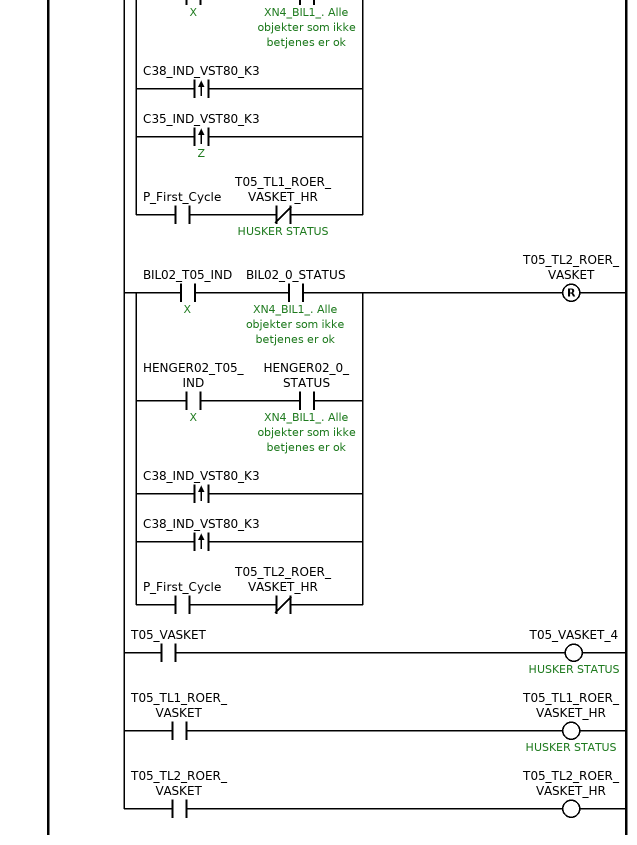
; [picture p936: NewProgram1 / T05_STATUS, rungs 1-1]
; rung 1: TANKOMRÅDET VASKET
LD P_On
OUT TR0
AND K3_TR23_TID_S
OUT TR1
LD C14_IND_VST80_K3  ; Z
OR C38_IND_VST80_K3
LD P_First_Cycle
AND T05_VASKET_4  ; HUSKER STATUS
ORLD
ANDLD
SET T05_VASKET
LD TR1
LD C38_IND_VST80_K3
OR C35_IND_VST80_K3  ; Z
LD P_First_Cycle
AND T05_TL1_ROER_VASKET_HR  ; HUSKER STATUS
ORLD
ANDLD
SET T05_TL1_ROER_VASKET
LD TR1
LD C38_IND_VST80_K3
OR C35_IND_VST80_K3  ; Z
LD P_First_Cycle
AND T05_TL2_ROER_VASKET_HR
ORLD
ANDLD
SET T05_TL2_ROER_VASKET
LD TR0
LD BIL01_T05_IND  ; X
AND BIL01_0_STATUS  ; XN4_BIL1_. Alle objekter som ikke betjenes er ok
LD HENGER01_T05_IND  ; X
AND HENGER01_0_STATUS  ; XN4_BIL1_. Alle objekter som ikke betjenes er ok
ORLD
LD BIL02_T05_IND  ; X
AND BIL02_0_STATUS  ; XN4_BIL1_. Alle objekter som ikke betjenes er ok
ORLD
LD HENGER02_T05_IND  ; X
AND HENGER02_0_STATUS  ; XN4_BIL1_. Alle objekter som ikke betjenes er ok
ORLD
@OR C38_IND_VST80_K3
@OR C14_IND_VST80_K3  ; Z
LD P_First_Cycle
ANDNOT T05_VASKET_4  ; HUSKER STATUS
ORLD
ANDLD
RSET T05_VASKET
LD TR0
LD BIL01_T05_IND  ; X
AND BIL01_0_STATUS  ; XN4_BIL1_. Alle objekter som ikke betjenes er ok
LD HENGER01_T05_IND  ; X
AND HENGER01_0_STATUS  ; XN4_BIL1_. Alle objekter som ikke betjenes er ok
ORLD
@OR C38_IND_VST80_K3
@OR C35_IND_VST80_K3  ; Z
LD P_First_Cycle
ANDNOT T05_TL1_ROER_VASKET_HR  ; HUSKER STATUS
ORLD
ANDLD
RSET T05_TL1_ROER_VASKET
LD TR0
LD BIL02_T05_IND  ; X
AND BIL02_0_STATUS  ; XN4_BIL1_. Alle objekter som ikke betjenes er ok
LD HENGER02_T05_IND  ; X
AND HENGER02_0_STATUS  ; XN4_BIL1_. Alle objekter som ikke betjenes er ok
ORLD
@OR C38_IND_VST80_K3
@OR C38_IND_VST80_K3
LD P_First_Cycle
ANDNOT T05_TL2_ROER_VASKET_HR
ORLD
ANDLD
RSET T05_TL2_ROER_VASKET
LD TR0
AND T05_VASKET
OUT T05_VASKET_4  ; HUSKER STATUS
LD TR0
AND T05_TL1_ROER_VASKET
OUT T05_TL1_ROER_VASKET_HR  ; HUSKER STATUS
LD TR0
AND T05_TL2_ROER_VASKET
OUT T05_TL2_ROER_VASKET_HR

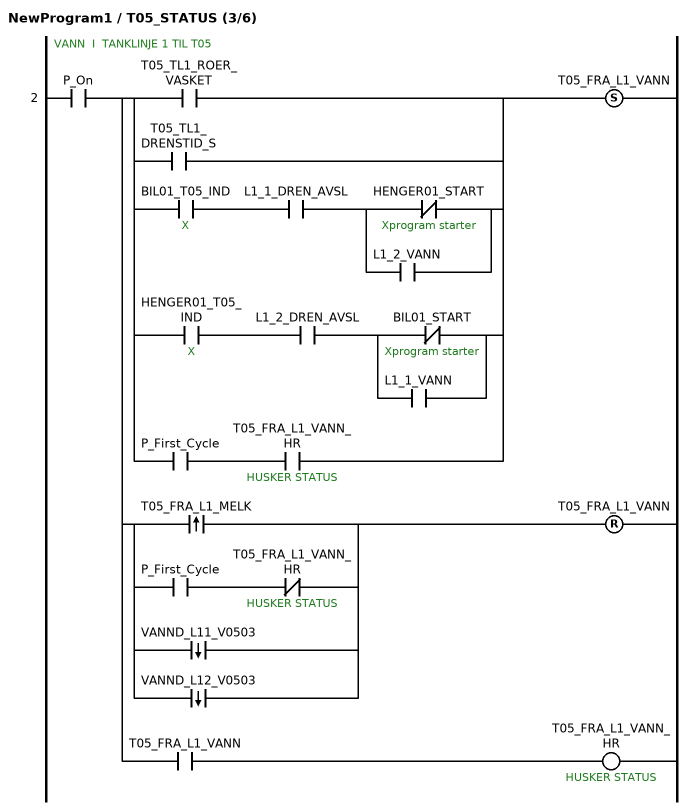
; rung 2: VANN  I  TANKLINJE 1 TIL T05
LD P_On
OUT TR0
LD T05_TL1_ROER_VASKET
OR T05_TL1_DRENSTID_S
LD BIL01_T05_IND  ; X
AND L1_1_DREN_AVSL
LDNOT HENGER01_START  ; Xprogram starter
OR L1_2_VANN
ANDLD
ORLD
LD HENGER01_T05_IND  ; X
AND L1_2_DREN_AVSL
LDNOT BIL01_START  ; Xprogram starter
OR L1_1_VANN
ANDLD
ORLD
LD P_First_Cycle
AND T05_FRA_L1_VANN_HR  ; HUSKER STATUS
ORLD
ANDLD
SET T05_FRA_L1_VANN
LD TR0
@LD T05_FRA_L1_MELK
LD P_First_Cycle
ANDNOT T05_FRA_L1_VANN_HR  ; HUSKER STATUS
ORLD
%OR VANND_L11_V0503
%OR VANND_L12_V0503
ANDLD
RSET T05_FRA_L1_VANN
LD TR0
AND T05_FRA_L1_VANN
OUT T05_FRA_L1_VANN_HR  ; HUSKER STATUS

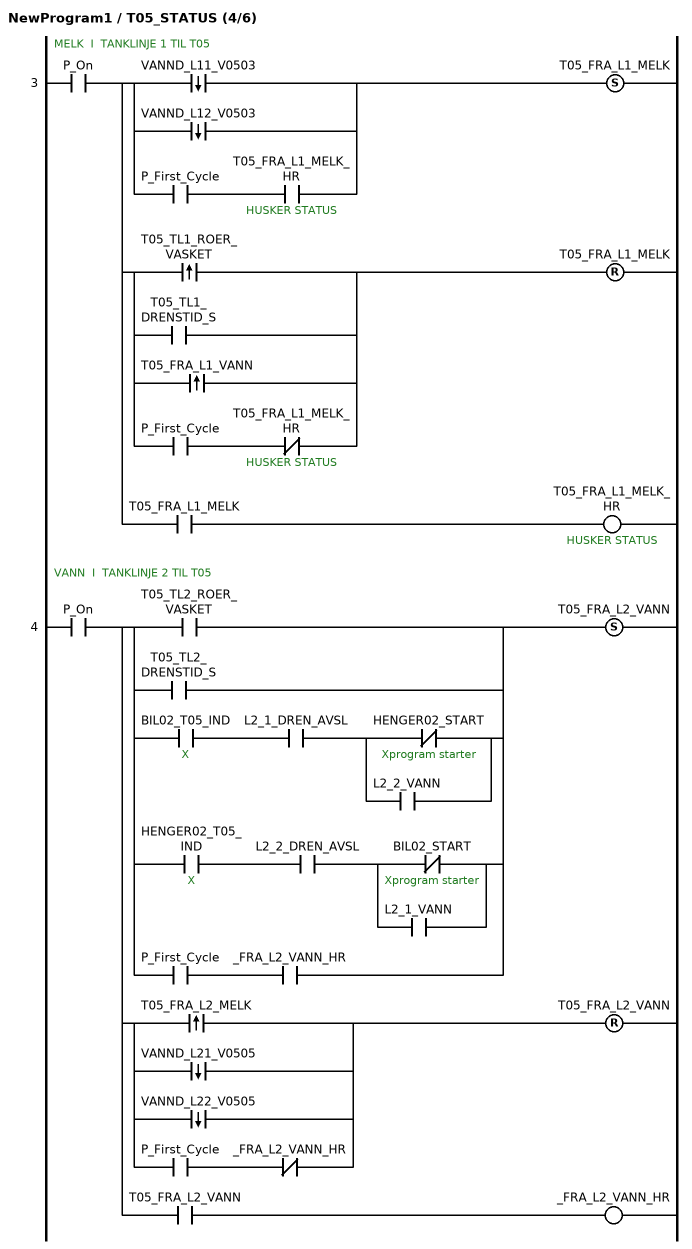
; rung 3: MELK  I  TANKLINJE 1 TIL T05
LD P_On
OUT TR0
%LD VANND_L11_V0503
%OR VANND_L12_V0503
LD P_First_Cycle
AND T05_FRA_L1_MELK_HR  ; HUSKER STATUS
ORLD
ANDLD
SET T05_FRA_L1_MELK
LD TR0
@LD T05_TL1_ROER_VASKET
OR T05_TL1_DRENSTID_S
@OR T05_FRA_L1_VANN
LD P_First_Cycle
ANDNOT T05_FRA_L1_MELK_HR  ; HUSKER STATUS
ORLD
ANDLD
RSET T05_FRA_L1_MELK
LD TR0
AND T05_FRA_L1_MELK
OUT T05_FRA_L1_MELK_HR  ; HUSKER STATUS
; rung 4: VANN  I  TANKLINJE 2 TIL T05
LD P_On
OUT TR0
LD T05_TL2_ROER_VASKET
OR T05_TL2_DRENSTID_S
LD BIL02_T05_IND  ; X
AND L2_1_DREN_AVSL
LDNOT HENGER02_START  ; Xprogram starter
OR L2_2_VANN
ANDLD
ORLD
LD HENGER02_T05_IND  ; X
AND L2_2_DREN_AVSL
LDNOT BIL02_START  ; Xprogram starter
OR L2_1_VANN
ANDLD
ORLD
LD P_First_Cycle
AND _FRA_L2_VANN_HR
ORLD
ANDLD
SET T05_FRA_L2_VANN
LD TR0
@LD T05_FRA_L2_MELK
%OR VANND_L21_V0505
%OR VANND_L22_V0505
LD P_First_Cycle
ANDNOT _FRA_L2_VANN_HR
ORLD
ANDLD
RSET T05_FRA_L2_VANN
LD TR0
AND T05_FRA_L2_VANN
OUT _FRA_L2_VANN_HR

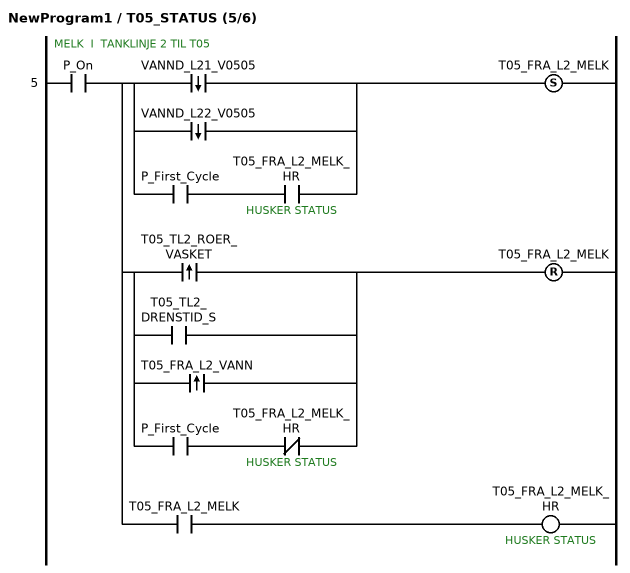
; rung 5: MELK  I  TANKLINJE 2 TIL T05
LD P_On
OUT TR0
%LD VANND_L21_V0505
%OR VANND_L22_V0505
LD P_First_Cycle
AND T05_FRA_L2_MELK_HR  ; HUSKER STATUS
ORLD
ANDLD
SET T05_FRA_L2_MELK
LD TR0
@LD T05_TL2_ROER_VASKET
OR T05_TL2_DRENSTID_S
@OR T05_FRA_L2_VANN
LD P_First_Cycle
ANDNOT T05_FRA_L2_MELK_HR  ; HUSKER STATUS
ORLD
ANDLD
RSET T05_FRA_L2_MELK
LD TR0
AND T05_FRA_L2_MELK
OUT T05_FRA_L2_MELK_HR  ; HUSKER STATUS

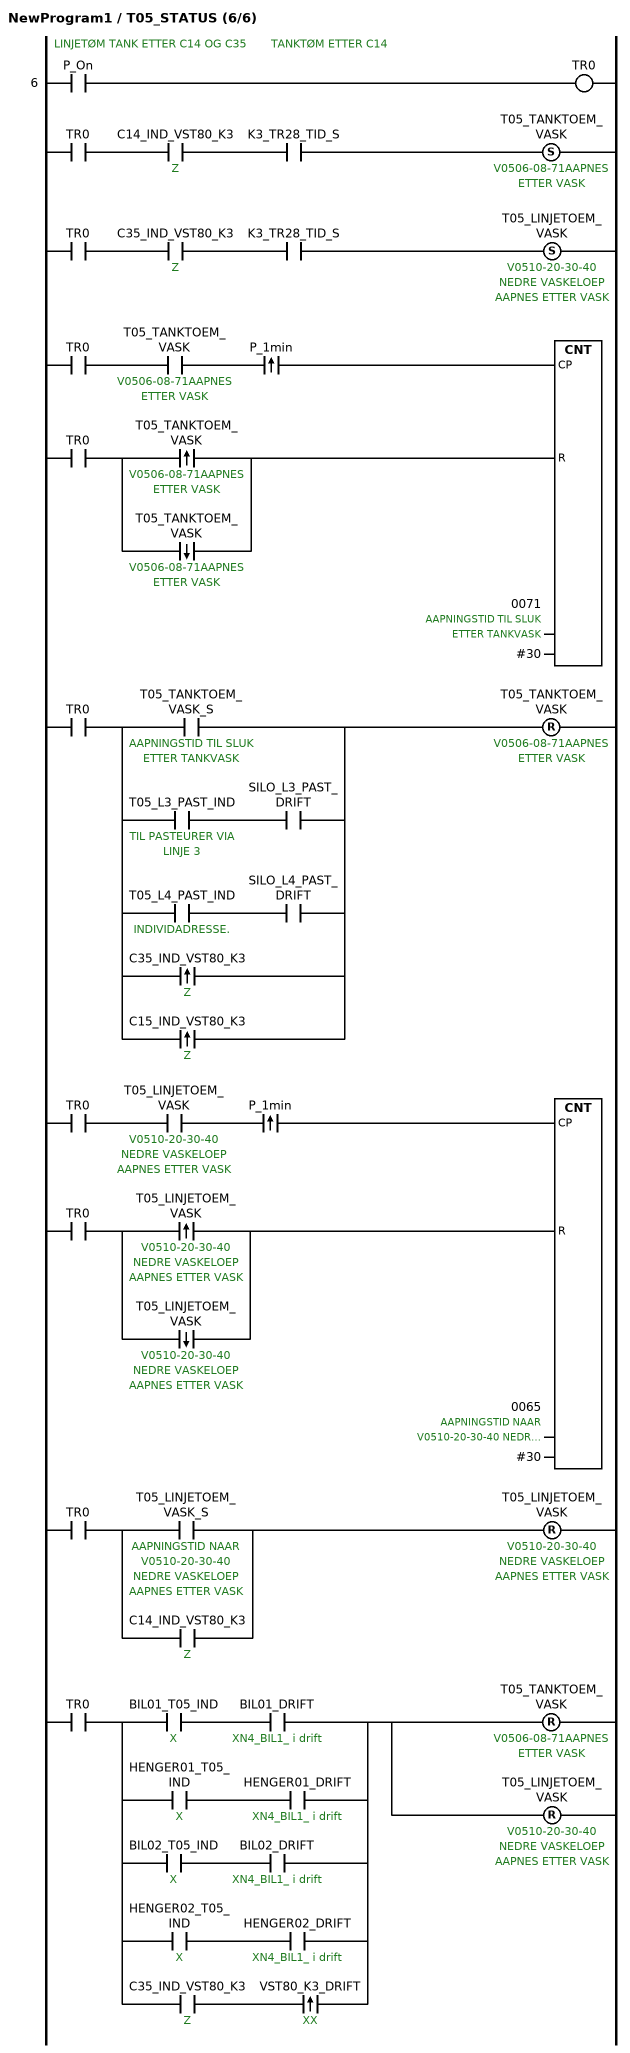
; rung 6: LINJETØM TANK ETTER C14 OG C35       TANKTØM ETTER C14
LD P_On
OUT TR0
AND C14_IND_VST80_K3  ; Z
AND K3_TR28_TID_S
SET T05_TANKTOEM_VASK  ; V0506-08-71AAPNES ETTER VASK
LD TR0
AND C35_IND_VST80_K3  ; Z
AND K3_TR28_TID_S
SET T05_LINJETOEM_VASK  ; V0510-20-30-40 NEDRE VASKELOEP AAPNES ETTER VASK
LD TR0
AND T05_TANKTOEM_VASK  ; V0506-08-71AAPNES ETTER VASK
@AND P_1min
LD TR0
@LD T05_TANKTOEM_VASK  ; V0506-08-71AAPNES ETTER VASK
%OR T05_TANKTOEM_VASK  ; V0506-08-71AAPNES ETTER VASK
ANDLD
CNT 0071 #30  ; AAPNINGSTID TIL SLUK ETTER TANKVASK
LD TR0
LD T05_TANKTOEM_VASK_S  ; AAPNINGSTID TIL SLUK ETTER TANKVASK
LD T05_L3_PAST_IND  ; TIL PASTEURER VIA LINJE 3
AND SILO_L3_PAST_DRIFT
ORLD
LD T05_L4_PAST_IND  ; INDIVIDADRESSE.
AND SILO_L4_PAST_DRIFT
ORLD
@OR C35_IND_VST80_K3  ; Z
@OR C15_IND_VST80_K3  ; Z
ANDLD
RSET T05_TANKTOEM_VASK  ; V0506-08-71AAPNES ETTER VASK
LD TR0
AND T05_LINJETOEM_VASK  ; V0510-20-30-40 NEDRE VASKELOEP AAPNES ETTER VASK
@AND P_1min
LD TR0
@LD T05_LINJETOEM_VASK  ; V0510-20-30-40 NEDRE VASKELOEP AAPNES ETTER VASK
%OR T05_LINJETOEM_VASK  ; V0510-20-30-40 NEDRE VASKELOEP AAPNES ETTER VASK
ANDLD
CNT 0065 #30  ; AAPNINGSTID NAAR V0510-20-30-40 NEDRE VASKELOEP AAPNES ETTER VASK
LD TR0
LD T05_LINJETOEM_VASK_S  ; AAPNINGSTID NAAR V0510-20-30-40 NEDRE VASKELOEP AAPNES ETTER VASK
OR C14_IND_VST80_K3  ; Z
ANDLD
RSET T05_LINJETOEM_VASK  ; V0510-20-30-40 NEDRE VASKELOEP AAPNES ETTER VASK
LD TR0
LD BIL01_T05_IND  ; X
AND BIL01_DRIFT  ; XN4_BIL1_ i drift
LD HENGER01_T05_IND  ; X
AND HENGER01_DRIFT  ; XN4_BIL1_ i drift
ORLD
LD BIL02_T05_IND  ; X
AND BIL02_DRIFT  ; XN4_BIL1_ i drift
ORLD
LD HENGER02_T05_IND  ; X
AND HENGER02_DRIFT  ; XN4_BIL1_ i drift
ORLD
LD C35_IND_VST80_K3  ; Z
@AND VST80_K3_DRIFT  ; XX
ORLD
ANDLD
RSET T05_TANKTOEM_VASK  ; V0506-08-71AAPNES ETTER VASK
RSET T05_LINJETOEM_VASK  ; V0510-20-30-40 NEDRE VASKELOEP AAPNES ETTER VASK
; rung 7: Ingen_kommentar_funnet

### Section T06_NIVÅ_HL_LL_FLOW

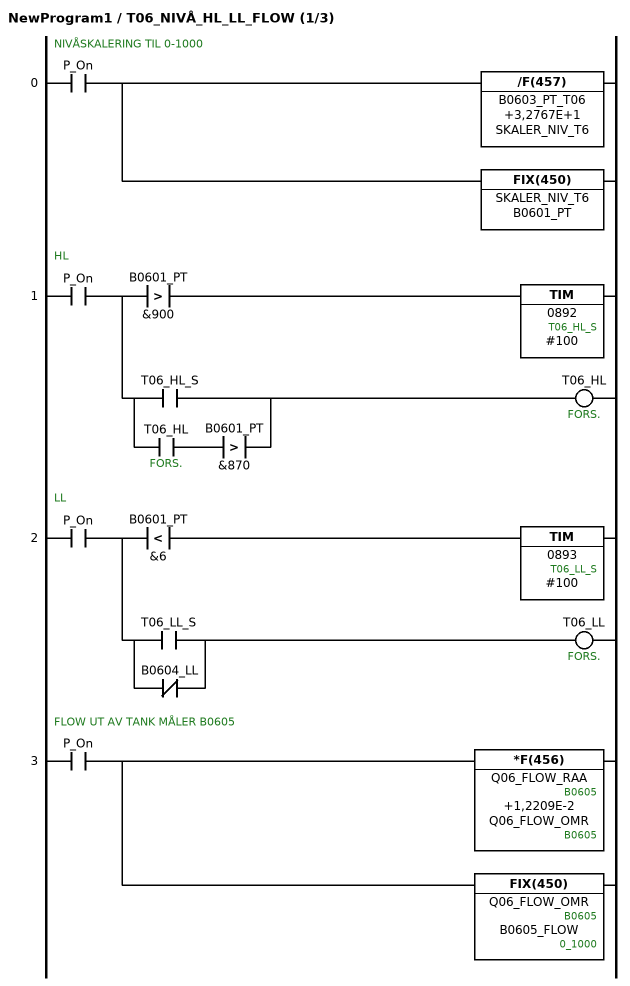
; rung 0: NIVÅSKALERING TIL 0-1000
LD P_On
/F(457) B0603_PT_T06 +3,2767E+1 SKALER_NIV_T6
FIX(450) SKALER_NIV_T6 B0601_PT
; rung 1: HL
LD P_On
OUT TR0
AND>(320) B0601_PT &900
TIM 0892 #100  ; T06_HL_S
LD TR0
LD T06_HL_S
LD T06_HL  ; FORS.
AND>(320) B0601_PT &870
ORLD
ANDLD
OUT T06_HL  ; FORS.
; rung 2: LL
LD P_On
OUT TR0
AND<(310) B0601_PT &6
TIM 0893 #100  ; T06_LL_S
LD TR0
LD T06_LL_S
ORNOT B0604_LL
ANDLD
OUT T06_LL  ; FORS.
; rung 3: FLOW UT AV TANK MÅLER B0605
LD P_On
*F(456) Q06_FLOW_RAA +1,2209E-2 Q06_FLOW_OMR  ; B0605  // Flow er gitt med verdiene 0-8000, som tilsvarer 0-80 m3
FIX(450) Q06_FLOW_OMR B0605_FLOW  ; B0605, 0_1000

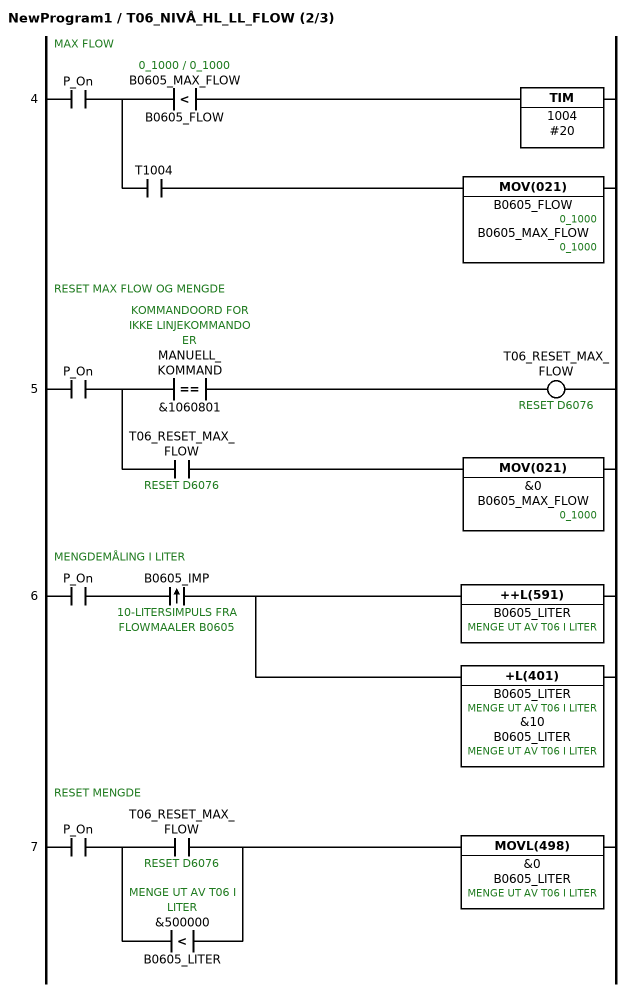
; rung 4: MAX FLOW
LD P_On
OUT TR0
AND<(310) B0605_MAX_FLOW B0605_FLOW  ; 0_1000
TIM 1004 #20
LD TR0
AND T1004
MOV(021) B0605_FLOW B0605_MAX_FLOW  ; 0_1000
; rung 5: RESET MAX FLOW OG MENGDE
LD P_On
OUT TR0
AND=L(301) MANUELL_KOMMAND &1060801  ; KOMMANDOORD FOR IKKE LINJEKOMMANDOER
OUT T06_RESET_MAX_FLOW  ; RESET D6076
LD TR0
AND T06_RESET_MAX_FLOW  ; RESET D6076
MOV(021) &0 B0605_MAX_FLOW  ; 0_1000
; rung 6: MENGDEMÅLING I LITER
LD P_On
@AND B0605_IMP  ; 10-LITERSIMPULS FRA FLOWMAALER B0605
++L(591) B0605_LITER  ; MENGE UT AV T06 I LITER
+L(401) B0605_LITER &10 B0605_LITER  ; MENGE UT AV T06 I LITER
; rung 7: RESET MENGDE
LD P_On
LD T06_RESET_MAX_FLOW  ; RESET D6076
OR<L(311) &500000 B0605_LITER  ; MENGE UT AV T06 I LITER
ANDLD
MOVL(498) &0 B0605_LITER  ; MENGE UT AV T06 I LITER

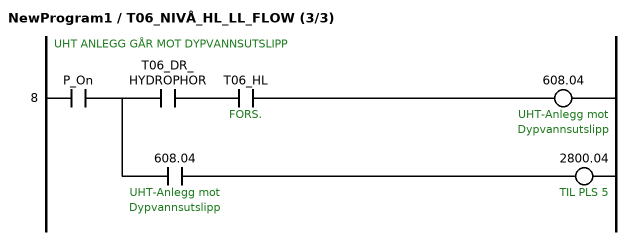
; rung 8: UHT ANLEGG GÅR MOT DYPVANNSUTSLIPP
LD P_On
OUT TR0
AND T06_DR_HYDROPHOR
AND T06_HL  ; FORS.
OUT 608.04  ; UHT-Anlegg mot Dypvannsutslipp
LD TR0
AND 608.04  ; UHT-Anlegg mot Dypvannsutslipp
OUT 2800.04  ; TIL PLS 5
; rung 9: Ingen_kommentar_funnet

### Section T06_TANKSPERR

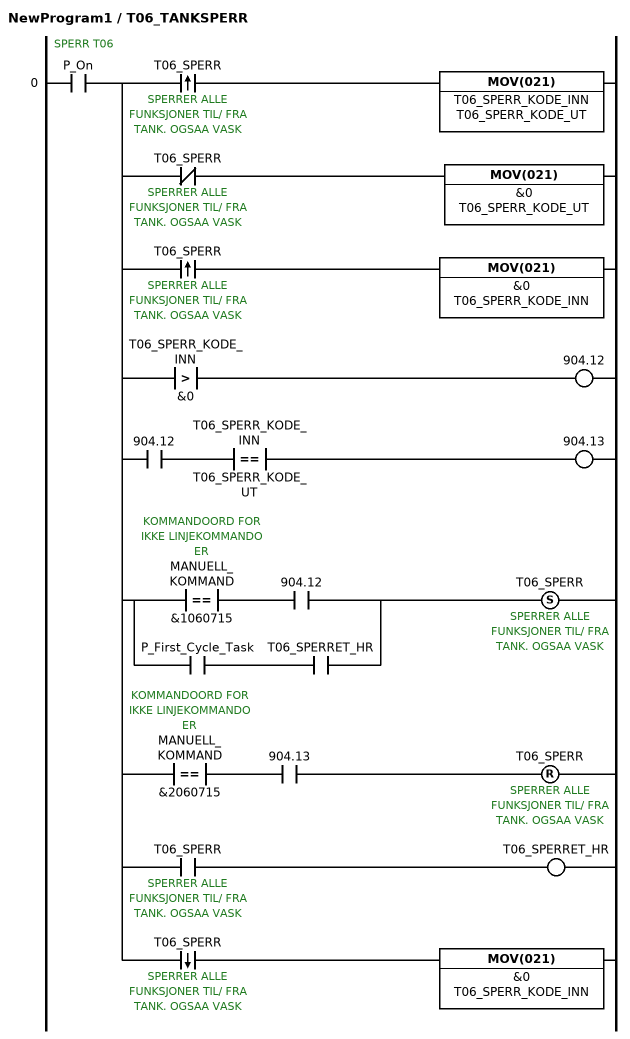
; rung 0: SPERR T06
LD P_On
OUT TR0
@AND T06_SPERR  ; SPERRER ALLE FUNKSJONER TIL/ FRA TANK. OGSAA VASK
MOV(021) T06_SPERR_KODE_INN T06_SPERR_KODE_UT
LD TR0
ANDNOT T06_SPERR  ; SPERRER ALLE FUNKSJONER TIL/ FRA TANK. OGSAA VASK
MOV(021) &0 T06_SPERR_KODE_UT
LD TR0
@AND T06_SPERR  ; SPERRER ALLE FUNKSJONER TIL/ FRA TANK. OGSAA VASK
MOV(021) &0 T06_SPERR_KODE_INN
LD TR0
AND>(320) T06_SPERR_KODE_INN &0
OUT 904.12
LD TR0
AND 904.12
AND=(300) T06_SPERR_KODE_INN T06_SPERR_KODE_UT
OUT 904.13
LD TR0
LD=L(301) MANUELL_KOMMAND &1060715  ; KOMMANDOORD FOR IKKE LINJEKOMMANDOER
AND 904.12
LD P_First_Cycle_Task
AND T06_SPERRET_HR
ORLD
ANDLD
SET T06_SPERR  ; SPERRER ALLE FUNKSJONER TIL/ FRA TANK. OGSAA VASK
LD TR0
AND=L(301) MANUELL_KOMMAND &2060715  ; KOMMANDOORD FOR IKKE LINJEKOMMANDOER
AND 904.13
RSET T06_SPERR  ; SPERRER ALLE FUNKSJONER TIL/ FRA TANK. OGSAA VASK
LD TR0
AND T06_SPERR  ; SPERRER ALLE FUNKSJONER TIL/ FRA TANK. OGSAA VASK
OUT T06_SPERRET_HR
LD TR0
%AND T06_SPERR  ; SPERRER ALLE FUNKSJONER TIL/ FRA TANK. OGSAA VASK
MOV(021) &0 T06_SPERR_KODE_INN
; rung 1: Ingen_kommentar_funnet

### Section T06_OBJEKTER

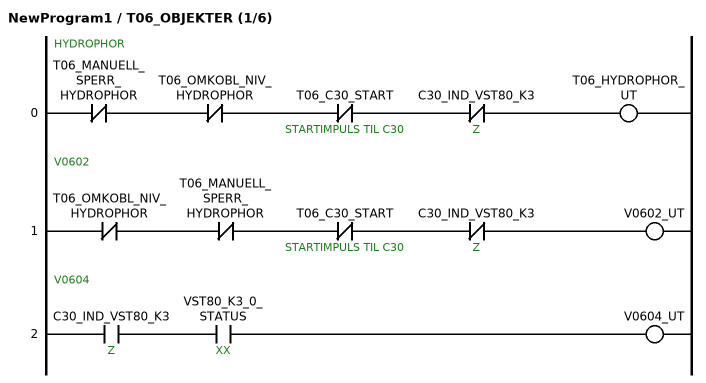
; rung 0: HYDROPHOR
LDNOT T06_MANUELL_SPERR_HYDROPHOR
ANDNOT T06_OMKOBL_NIV_HYDROPHOR
ANDNOT T06_C30_START  ; STARTIMPULS TIL C30
ANDNOT C30_IND_VST80_K3  ; Z
OUT T06_HYDROPHOR_UT
; rung 1: V0602
LDNOT T06_OMKOBL_NIV_HYDROPHOR
ANDNOT T06_MANUELL_SPERR_HYDROPHOR
ANDNOT T06_C30_START  ; STARTIMPULS TIL C30
ANDNOT C30_IND_VST80_K3  ; Z
OUT V0602_UT
; rung 2: V0604
LD C30_IND_VST80_K3  ; Z
AND VST80_K3_0_STATUS  ; XX
OUT V0604_UT

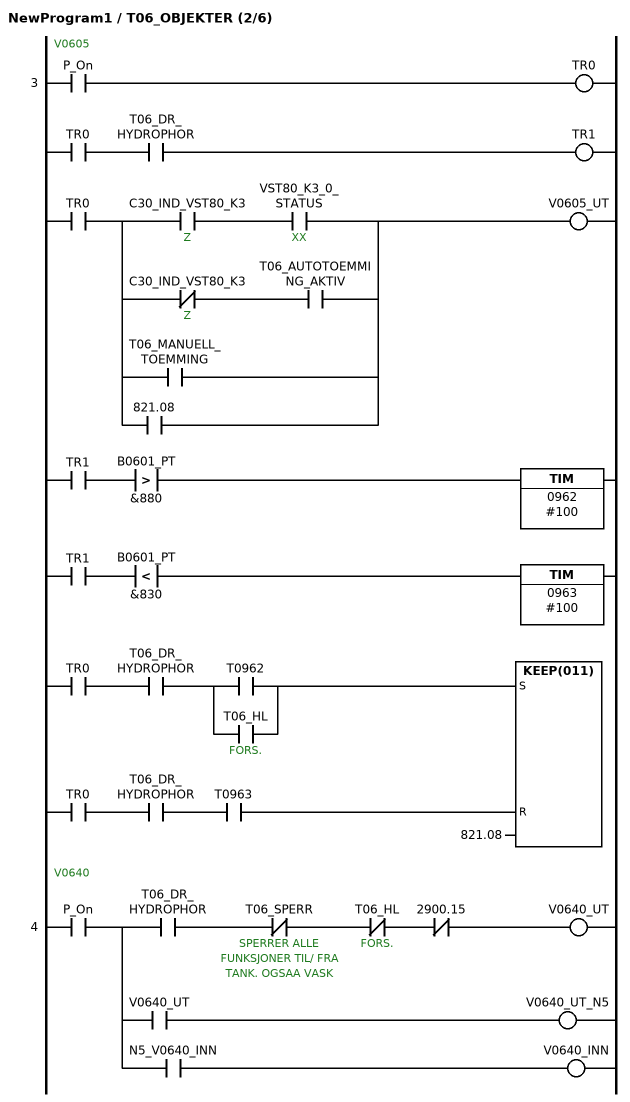
; rung 3: V0605
LD P_On
OUT TR0
LD C30_IND_VST80_K3  ; Z
AND VST80_K3_0_STATUS  ; XX
LDNOT C30_IND_VST80_K3  ; Z
AND T06_AUTOTOEMMING_AKTIV
ORLD
OR T06_MANUELL_TOEMMING
OR 821.08
ANDLD
OUT V0605_UT
LD TR0
AND T06_DR_HYDROPHOR
OUT TR1
AND>(320) B0601_PT &880
TIM 0962 #100
LD TR1
AND<(310) B0601_PT &830
TIM 0963 #100
LD TR0
AND T06_DR_HYDROPHOR
LD T0962
OR T06_HL  ; FORS.
ANDLD
LD TR0
AND T06_DR_HYDROPHOR
AND T0963
KEEP(011) 821.08
; rung 4: V0640
LD P_On
OUT TR0
AND T06_DR_HYDROPHOR
ANDNOT T06_SPERR  ; SPERRER ALLE FUNKSJONER TIL/ FRA TANK. OGSAA VASK
ANDNOT T06_HL  ; FORS.
ANDNOT 2900.15
OUT V0640_UT
LD TR0
AND V0640_UT
OUT V0640_UT_N5
LD TR0
AND N5_V0640_INN
OUT V0640_INN

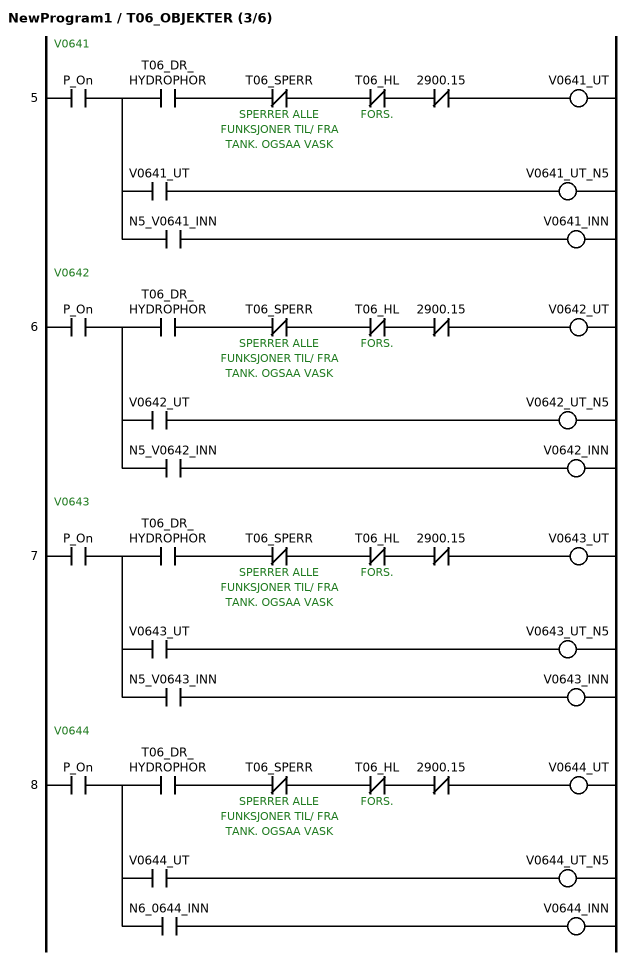
; rung 5: V0641
LD P_On
OUT TR0
AND T06_DR_HYDROPHOR
ANDNOT T06_SPERR  ; SPERRER ALLE FUNKSJONER TIL/ FRA TANK. OGSAA VASK
ANDNOT T06_HL  ; FORS.
ANDNOT 2900.15
OUT V0641_UT
LD TR0
AND V0641_UT
OUT V0641_UT_N5
LD TR0
AND N5_V0641_INN
OUT V0641_INN
; rung 6: V0642
LD P_On
OUT TR0
AND T06_DR_HYDROPHOR
ANDNOT T06_SPERR  ; SPERRER ALLE FUNKSJONER TIL/ FRA TANK. OGSAA VASK
ANDNOT T06_HL  ; FORS.
ANDNOT 2900.15
OUT V0642_UT
LD TR0
AND V0642_UT
OUT V0642_UT_N5
LD TR0
AND N5_V0642_INN
OUT V0642_INN
; rung 7: V0643
LD P_On
OUT TR0
AND T06_DR_HYDROPHOR
ANDNOT T06_SPERR  ; SPERRER ALLE FUNKSJONER TIL/ FRA TANK. OGSAA VASK
ANDNOT T06_HL  ; FORS.
ANDNOT 2900.15
OUT V0643_UT
LD TR0
AND V0643_UT
OUT V0643_UT_N5
LD TR0
AND N5_V0643_INN
OUT V0643_INN
; rung 8: V0644
LD P_On
OUT TR0
AND T06_DR_HYDROPHOR
ANDNOT T06_SPERR  ; SPERRER ALLE FUNKSJONER TIL/ FRA TANK. OGSAA VASK
ANDNOT T06_HL  ; FORS.
ANDNOT 2900.15
OUT V0644_UT
LD TR0
AND V0644_UT
OUT V0644_UT_N5
LD TR0
AND N6_0644_INN
OUT V0644_INN

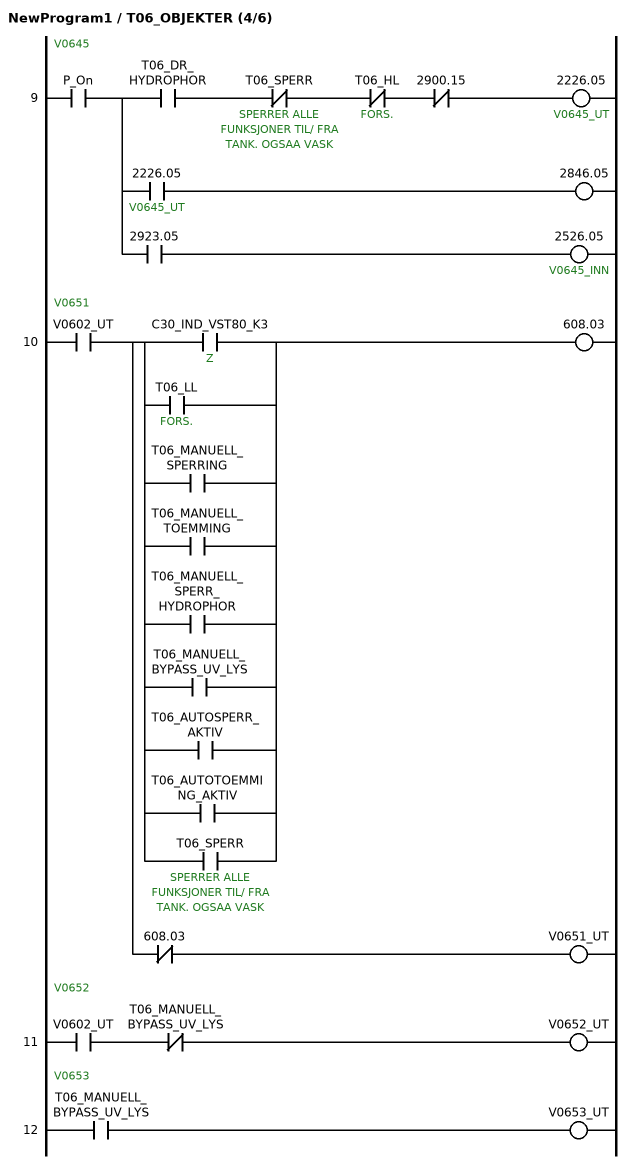
; rung 9: V0645
LD P_On
OUT TR0
AND T06_DR_HYDROPHOR
ANDNOT T06_SPERR  ; SPERRER ALLE FUNKSJONER TIL/ FRA TANK. OGSAA VASK
ANDNOT T06_HL  ; FORS.
ANDNOT 2900.15
OUT 2226.05  ; V0645_UT
LD TR0
AND 2226.05  ; V0645_UT
OUT 2846.05
LD TR0
AND 2923.05
OUT 2526.05  ; V0645_INN
; rung 10: V0651
LD V0602_UT
OUT TR0
LD C30_IND_VST80_K3  ; Z
OR T06_LL  ; FORS.
OR T06_MANUELL_SPERRING
OR T06_MANUELL_TOEMMING
OR T06_MANUELL_SPERR_HYDROPHOR
OR T06_MANUELL_BYPASS_UV_LYS
OR T06_AUTOSPERR_AKTIV
OR T06_AUTOTOEMMING_AKTIV
OR T06_SPERR  ; SPERRER ALLE FUNKSJONER TIL/ FRA TANK. OGSAA VASK
ANDLD
OUT 608.03
LD TR0
ANDNOT 608.03
OUT V0651_UT
; rung 11: V0652
LD V0602_UT
ANDNOT T06_MANUELL_BYPASS_UV_LYS
OUT V0652_UT
; rung 12: V0653
LD T06_MANUELL_BYPASS_UV_LYS
OUT V0653_UT

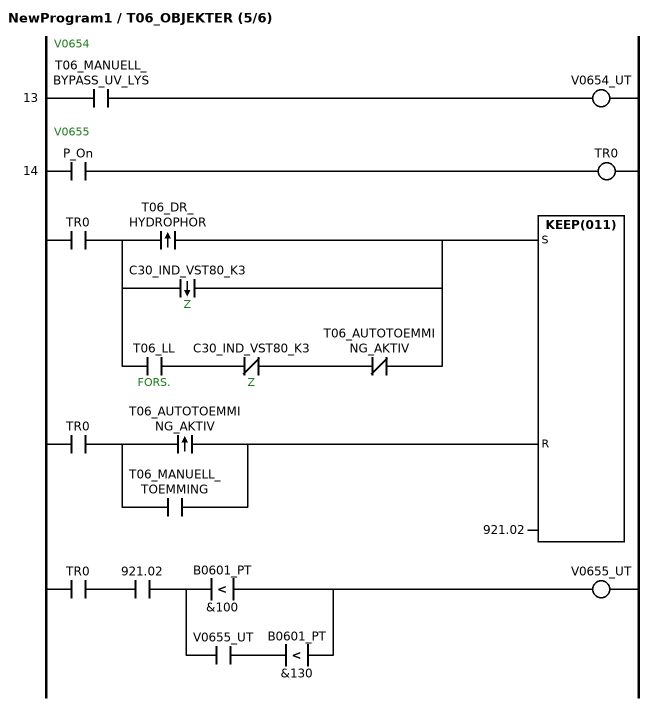
; rung 13: V0654
LD T06_MANUELL_BYPASS_UV_LYS
OUT V0654_UT
; rung 14: V0655
LD P_On
OUT TR0
@LD T06_DR_HYDROPHOR
%OR C30_IND_VST80_K3  ; Z
LD T06_LL  ; FORS.
ANDNOT C30_IND_VST80_K3  ; Z
ANDNOT T06_AUTOTOEMMING_AKTIV
ORLD
ANDLD
LD TR0
@LD T06_AUTOTOEMMING_AKTIV
OR T06_MANUELL_TOEMMING
ANDLD
KEEP(011) 921.02
LD TR0
AND 921.02
LD<(310) B0601_PT &100
LD V0655_UT
AND<(310) B0601_PT &130
ORLD
ANDLD
OUT V0655_UT

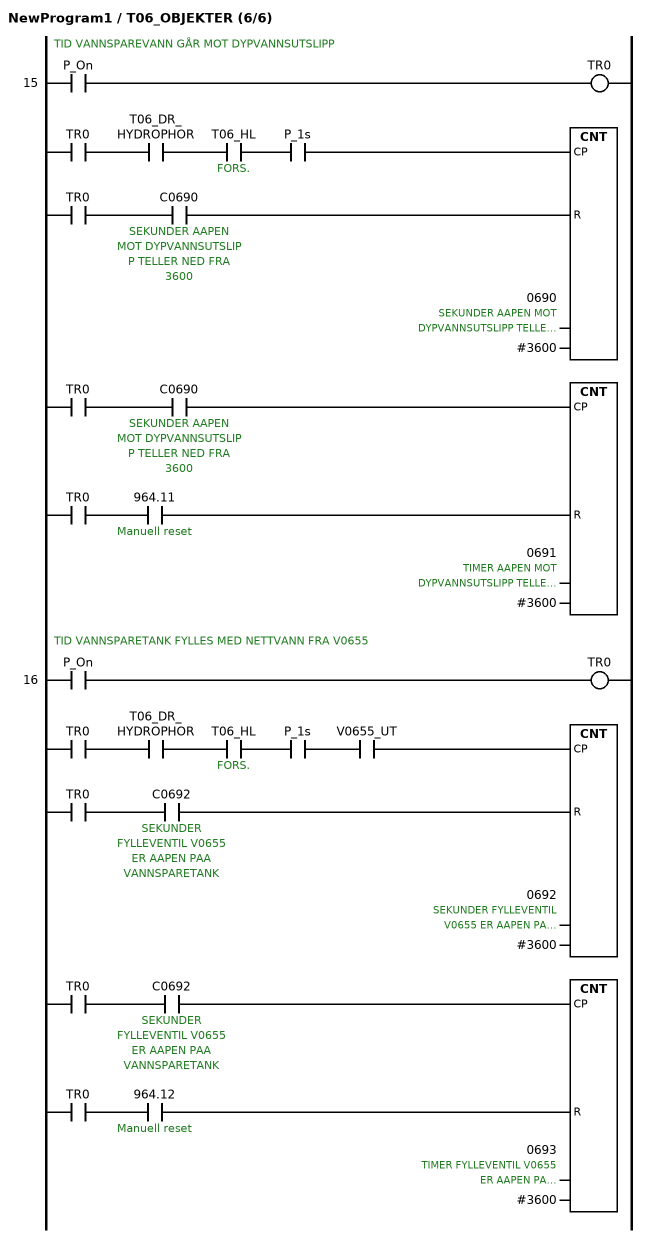
; rung 15: TID VANNSPAREVANN GÅR MOT DYPVANNSUTSLIPP
LD P_On
OUT TR0
AND T06_DR_HYDROPHOR
AND T06_HL  ; FORS.
AND P_1s
LD TR0
AND C0690  ; SEKUNDER AAPEN MOT DYPVANNSUTSLIPP TELLER NED FRA 3600
CNT 0690 #3600  ; SEKUNDER AAPEN MOT DYPVANNSUTSLIPP TELLER NED FRA 3600
LD TR0
AND C0690  ; SEKUNDER AAPEN MOT DYPVANNSUTSLIPP TELLER NED FRA 3600
LD TR0
AND 964.11  ; Manuell reset
CNT 0691 #3600  ; TIMER AAPEN MOT DYPVANNSUTSLIPP TELLER NED FRA 3600
; rung 16: TID VANNSPARETANK FYLLES MED NETTVANN FRA V0655
LD P_On
OUT TR0
AND T06_DR_HYDROPHOR
AND T06_HL  ; FORS.
AND P_1s
AND V0655_UT
LD TR0
AND C0692  ; SEKUNDER FYLLEVENTIL V0655 ER AAPEN PAA VANNSPARETANK
CNT 0692 #3600  ; SEKUNDER FYLLEVENTIL V0655 ER AAPEN PAA VANNSPARETANK
LD TR0
AND C0692  ; SEKUNDER FYLLEVENTIL V0655 ER AAPEN PAA VANNSPARETANK
LD TR0
AND 964.12  ; Manuell reset
CNT 0693 #3600  ; TIMER FYLLEVENTIL V0655 ER AAPEN PAA VANNSPARETANK
; rung 17: Ingen_kommentar_funnet

### Section T06_FUNKSJONSPERRER

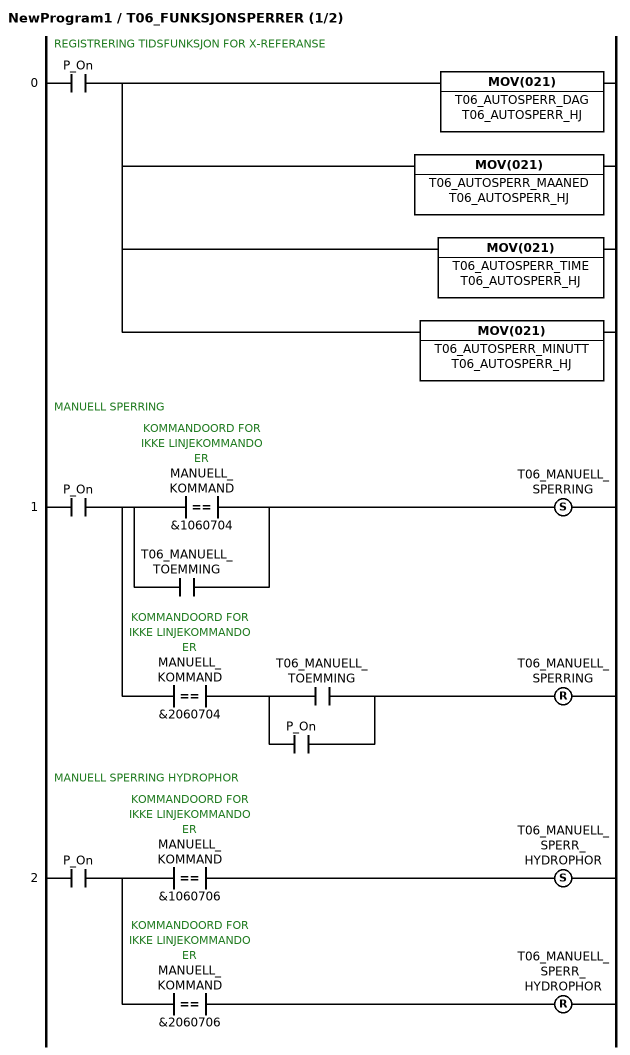
; rung 0: REGISTRERING TIDSFUNKSJON FOR X-REFERANSE
LD P_On
MOV(021) T06_AUTOSPERR_DAG T06_AUTOSPERR_HJ
MOV(021) T06_AUTOSPERR_MAANED T06_AUTOSPERR_HJ
MOV(021) T06_AUTOSPERR_TIME T06_AUTOSPERR_HJ
MOV(021) T06_AUTOSPERR_MINUTT T06_AUTOSPERR_HJ
; rung 1: MANUELL SPERRING
LD P_On
OUT TR0
LD=L(301) MANUELL_KOMMAND &1060704  ; KOMMANDOORD FOR IKKE LINJEKOMMANDOER
OR T06_MANUELL_TOEMMING
ANDLD
SET T06_MANUELL_SPERRING
LD TR0
AND=L(301) MANUELL_KOMMAND &2060704  ; KOMMANDOORD FOR IKKE LINJEKOMMANDOER
LD T06_MANUELL_TOEMMING
OR P_On
ANDLD
RSET T06_MANUELL_SPERRING
; rung 2: MANUELL SPERRING HYDROPHOR
LD P_On
OUT TR0
AND=L(301) MANUELL_KOMMAND &1060706  ; KOMMANDOORD FOR IKKE LINJEKOMMANDOER
SET T06_MANUELL_SPERR_HYDROPHOR
LD TR0
AND=L(301) MANUELL_KOMMAND &2060706  ; KOMMANDOORD FOR IKKE LINJEKOMMANDOER
RSET T06_MANUELL_SPERR_HYDROPHOR

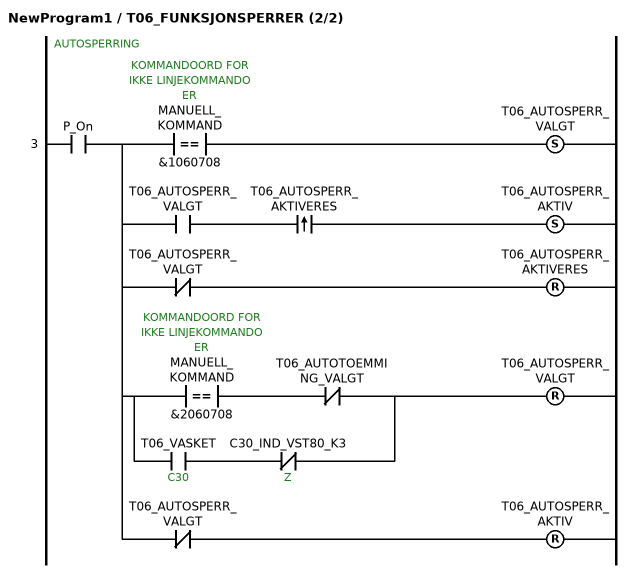
; rung 3: AUTOSPERRING
LD P_On
OUT TR0
AND=L(301) MANUELL_KOMMAND &1060708  ; KOMMANDOORD FOR IKKE LINJEKOMMANDOER
SET T06_AUTOSPERR_VALGT
LD TR0
AND T06_AUTOSPERR_VALGT
@AND T06_AUTOSPERR_AKTIVERES
SET T06_AUTOSPERR_AKTIV
LD TR0
ANDNOT T06_AUTOSPERR_VALGT
RSET T06_AUTOSPERR_AKTIVERES
LD TR0
LD=L(301) MANUELL_KOMMAND &2060708  ; KOMMANDOORD FOR IKKE LINJEKOMMANDOER
ANDNOT T06_AUTOTOEMMING_VALGT
LD T06_VASKET  ; C30
ANDNOT C30_IND_VST80_K3  ; Z
ORLD
ANDLD
RSET T06_AUTOSPERR_VALGT
LD TR0
ANDNOT T06_AUTOSPERR_VALGT
RSET T06_AUTOSPERR_AKTIV
; rung 4: Ingen_kommentar_funnet

### Section T06_TØMMEFUNKSJONER

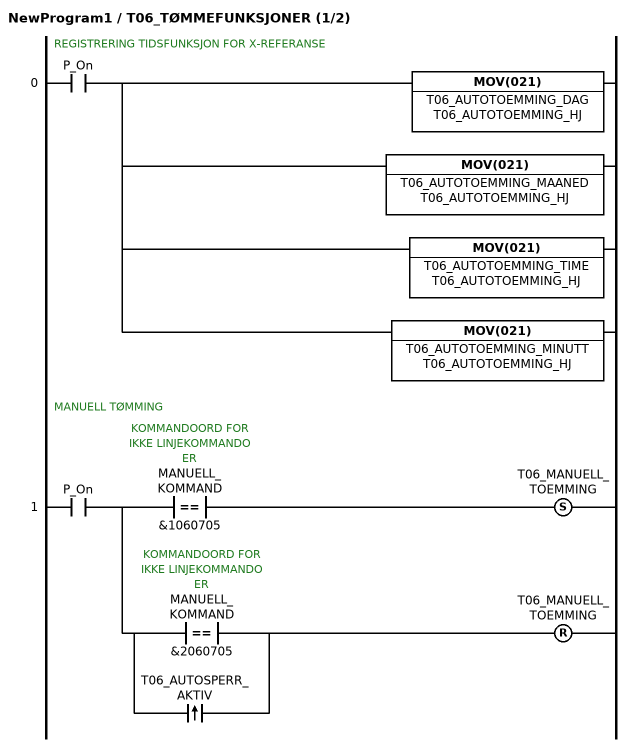
; rung 0: REGISTRERING TIDSFUNKSJON FOR X-REFERANSE
LD P_On
MOV(021) T06_AUTOTOEMMING_DAG T06_AUTOTOEMMING_HJ
MOV(021) T06_AUTOTOEMMING_MAANED T06_AUTOTOEMMING_HJ
MOV(021) T06_AUTOTOEMMING_TIME T06_AUTOTOEMMING_HJ
MOV(021) T06_AUTOTOEMMING_MINUTT T06_AUTOTOEMMING_HJ
; rung 1: MANUELL TØMMING
LD P_On
OUT TR0
AND=L(301) MANUELL_KOMMAND &1060705  ; KOMMANDOORD FOR IKKE LINJEKOMMANDOER
SET T06_MANUELL_TOEMMING
LD TR0
LD=L(301) MANUELL_KOMMAND &2060705  ; KOMMANDOORD FOR IKKE LINJEKOMMANDOER
@OR T06_AUTOSPERR_AKTIV
ANDLD
RSET T06_MANUELL_TOEMMING

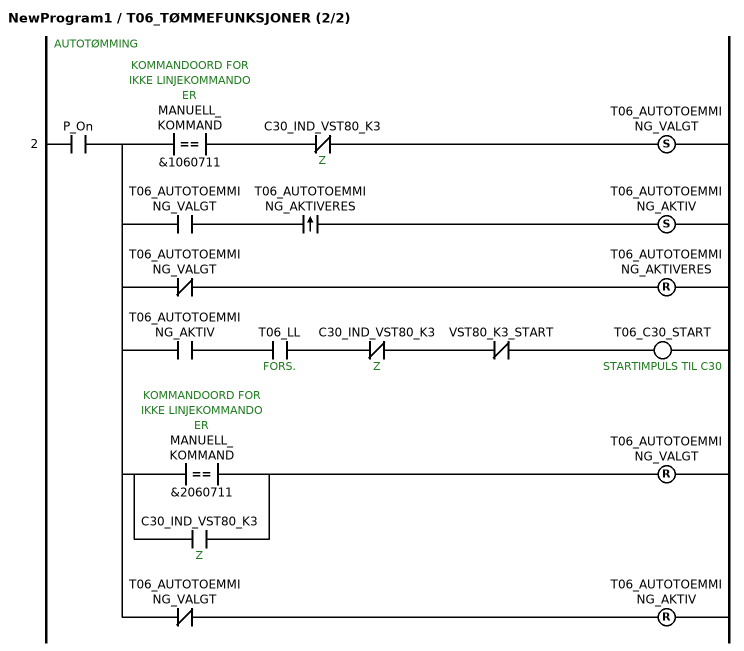
; rung 2: AUTOTØMMING
LD P_On
OUT TR0
AND=L(301) MANUELL_KOMMAND &1060711  ; KOMMANDOORD FOR IKKE LINJEKOMMANDOER
ANDNOT C30_IND_VST80_K3  ; Z
SET T06_AUTOTOEMMING_VALGT
LD TR0
AND T06_AUTOTOEMMING_VALGT
@AND T06_AUTOTOEMMING_AKTIVERES
SET T06_AUTOTOEMMING_AKTIV
LD TR0
ANDNOT T06_AUTOTOEMMING_VALGT
RSET T06_AUTOTOEMMING_AKTIVERES
LD TR0
AND T06_AUTOTOEMMING_AKTIV
AND T06_LL  ; FORS.
ANDNOT C30_IND_VST80_K3  ; Z
ANDNOT VST80_K3_START
OUT T06_C30_START  ; STARTIMPULS TIL C30
LD TR0
LD=L(301) MANUELL_KOMMAND &2060711  ; KOMMANDOORD FOR IKKE LINJEKOMMANDOER
OR C30_IND_VST80_K3  ; Z
ANDLD
RSET T06_AUTOTOEMMING_VALGT
LD TR0
ANDNOT T06_AUTOTOEMMING_VALGT
RSET T06_AUTOTOEMMING_AKTIV
; rung 3: Ingen_kommentar_funnet

### Section T06_FUNKSJONER

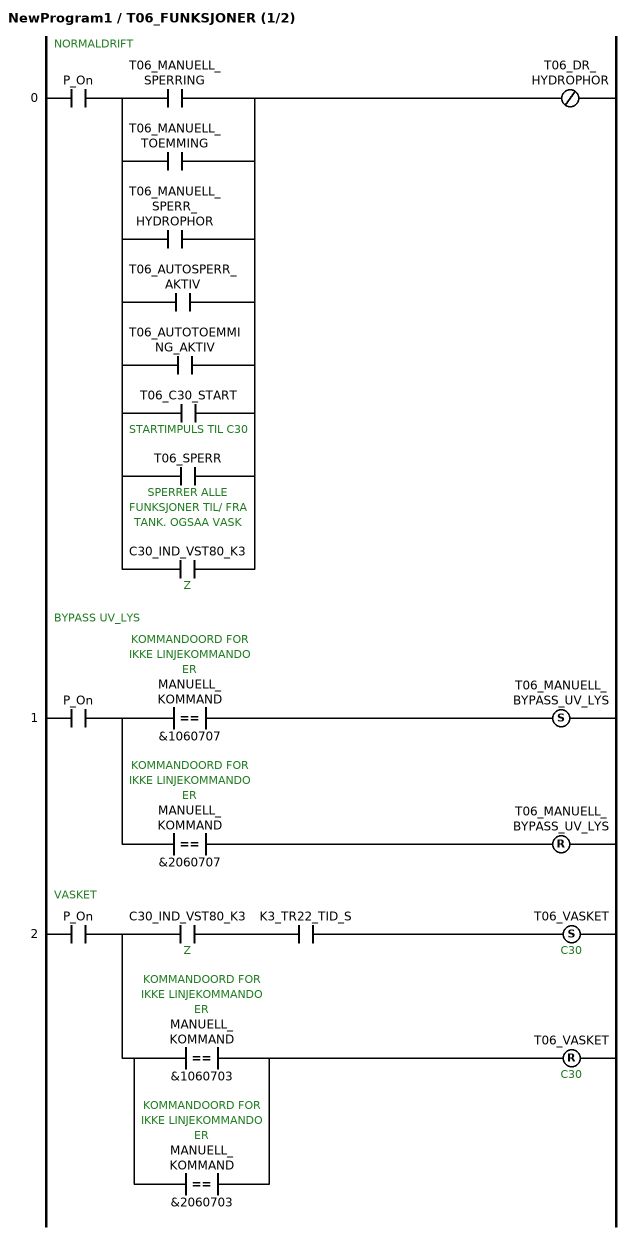
; rung 0: NORMALDRIFT
LD P_On
LD T06_MANUELL_SPERRING
OR T06_MANUELL_TOEMMING
OR T06_MANUELL_SPERR_HYDROPHOR
OR T06_AUTOSPERR_AKTIV
OR T06_AUTOTOEMMING_AKTIV
OR T06_C30_START  ; STARTIMPULS TIL C30
OR T06_SPERR  ; SPERRER ALLE FUNKSJONER TIL/ FRA TANK. OGSAA VASK
OR C30_IND_VST80_K3  ; Z
ANDLD
OUTNOT T06_DR_HYDROPHOR
; rung 1: BYPASS UV_LYS
LD P_On
OUT TR0
AND=L(301) MANUELL_KOMMAND &1060707  ; KOMMANDOORD FOR IKKE LINJEKOMMANDOER
SET T06_MANUELL_BYPASS_UV_LYS
LD TR0
AND=L(301) MANUELL_KOMMAND &2060707  ; KOMMANDOORD FOR IKKE LINJEKOMMANDOER
RSET T06_MANUELL_BYPASS_UV_LYS
; rung 2: VASKET
LD P_On
OUT TR0
AND C30_IND_VST80_K3  ; Z
AND K3_TR22_TID_S
SET T06_VASKET  ; C30
LD TR0
LD=L(301) MANUELL_KOMMAND &1060703  ; KOMMANDOORD FOR IKKE LINJEKOMMANDOER
OR=L(301) MANUELL_KOMMAND &2060703  ; KOMMANDOORD FOR IKKE LINJEKOMMANDOER
ANDLD
RSET T06_VASKET  ; C30

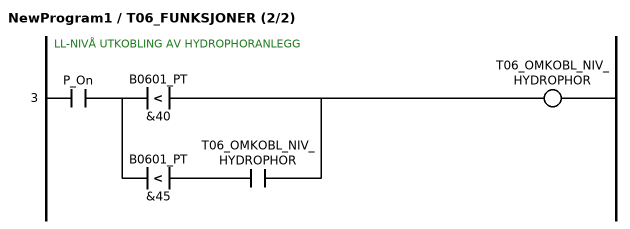
; rung 3: LL-NIVÅ UTKOBLING AV HYDROPHORANLEGG
LD P_On
LD<L(311) B0601_PT &40
LD<L(311) B0601_PT &45
AND T06_OMKOBL_NIV_HYDROPHOR
ORLD
ANDLD
OUT T06_OMKOBL_NIV_HYDROPHOR
; rung 4: Ingen_kommentar_funnet

### Section T07_01

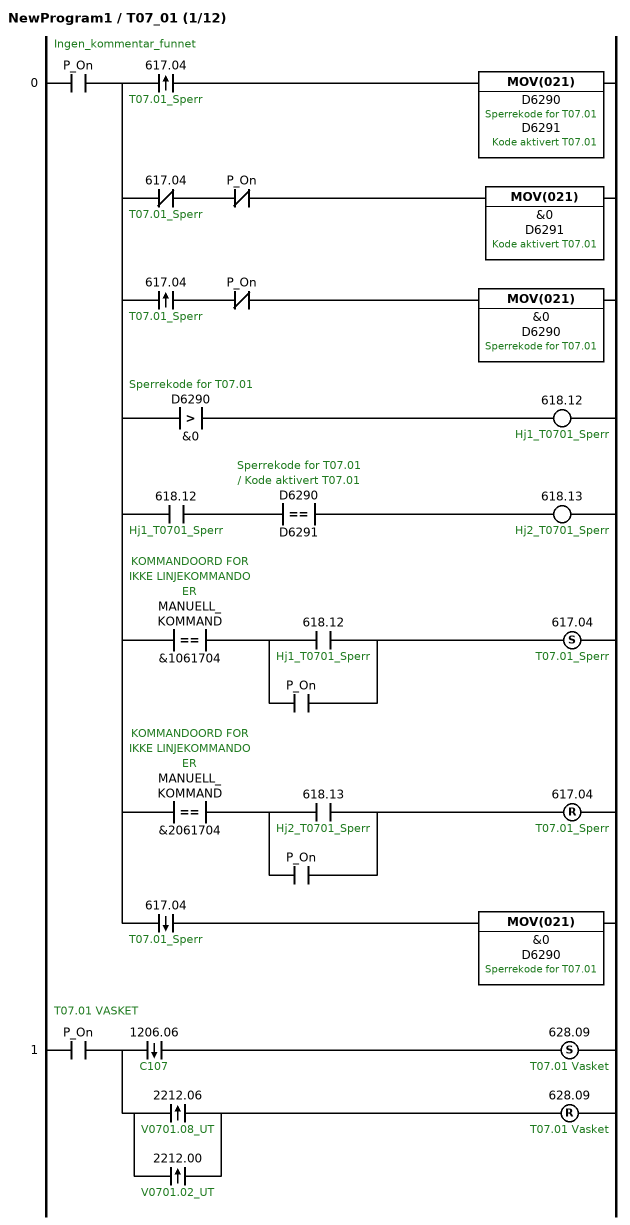
; rung 0: Ingen_kommentar_funnet
LD P_On
OUT TR0
@AND 617.04  ; T07.01_Sperr
MOV(021) D6290 D6291  ; Sperrekode for T07.01, Kode aktivert T07.01
LD TR0
ANDNOT 617.04  ; T07.01_Sperr
ANDNOT P_On
MOV(021) &0 D6291  ; Kode aktivert T07.01
LD TR0
@AND 617.04  ; T07.01_Sperr
ANDNOT P_On
MOV(021) &0 D6290  ; Sperrekode for T07.01
LD TR0
AND>(320) D6290 &0  ; Sperrekode for T07.01
OUT 618.12  ; Hj1_T0701_Sperr
LD TR0
AND 618.12  ; Hj1_T0701_Sperr
AND=(300) D6290 D6291  ; Sperrekode for T07.01, Kode aktivert T07.01
OUT 618.13  ; Hj2_T0701_Sperr
LD TR0
AND=L(301) MANUELL_KOMMAND &1061704  ; KOMMANDOORD FOR IKKE LINJEKOMMANDOER
LD 618.12  ; Hj1_T0701_Sperr
OR P_On
ANDLD
SET 617.04  ; T07.01_Sperr
LD TR0
AND=L(301) MANUELL_KOMMAND &2061704  ; KOMMANDOORD FOR IKKE LINJEKOMMANDOER
LD 618.13  ; Hj2_T0701_Sperr
OR P_On
ANDLD
RSET 617.04  ; T07.01_Sperr
LD TR0
%AND 617.04  ; T07.01_Sperr
MOV(021) &0 D6290  ; Sperrekode for T07.01
; rung 1: T07.01 VASKET
LD P_On
OUT TR0
%AND 1206.06  ; C107
SET 628.09  ; T07.01 Vasket
LD TR0
@LD 2212.06  ; V0701.08_UT
@OR 2212.00  ; V0701.02_UT
ANDLD
RSET 628.09  ; T07.01 Vasket

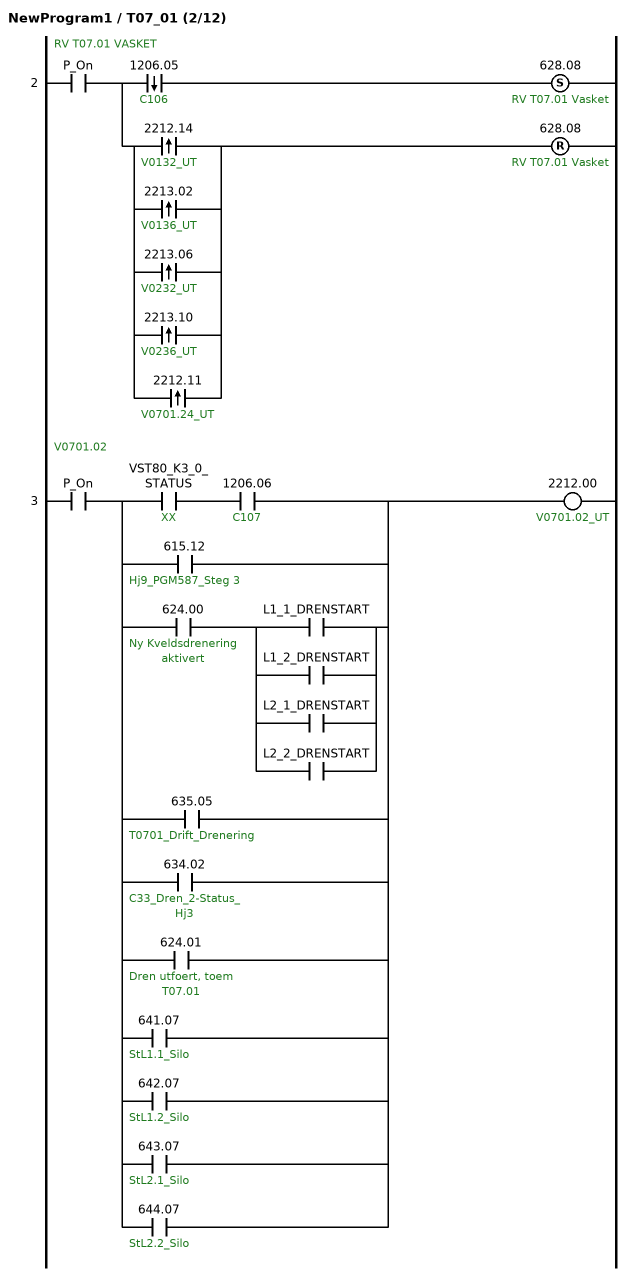
; rung 2: RV T07.01 VASKET
LD P_On
OUT TR0
%AND 1206.05  ; C106
SET 628.08  ; RV T07.01 Vasket
LD TR0
@LD 2212.14  ; V0132_UT
@OR 2213.02  ; V0136_UT
@OR 2213.06  ; V0232_UT
@OR 2213.10  ; V0236_UT
@OR 2212.11  ; V0701.24_UT
ANDLD
RSET 628.08  ; RV T07.01 Vasket
; rung 3: V0701.02
LD P_On
LD VST80_K3_0_STATUS  ; XX
AND 1206.06  ; C107
OR 615.12  ; Hj9_PGM587_Steg 3
LD 624.00  ; Ny Kveldsdrenering aktivert
LD L1_1_DRENSTART
OR L1_2_DRENSTART
OR L2_1_DRENSTART
OR L2_2_DRENSTART
ANDLD
ORLD
OR 635.05  ; T0701_Drift_Drenering
OR 634.02  ; C33_Dren_2-Status_Hj3
OR 624.01  ; Dren utfoert, toem T07.01
OR 641.07  ; StL1.1_Silo
OR 642.07  ; StL1.2_Silo
OR 643.07  ; StL2.1_Silo
OR 644.07  ; StL2.2_Silo
ANDLD
OUT 2212.00  ; V0701.02_UT

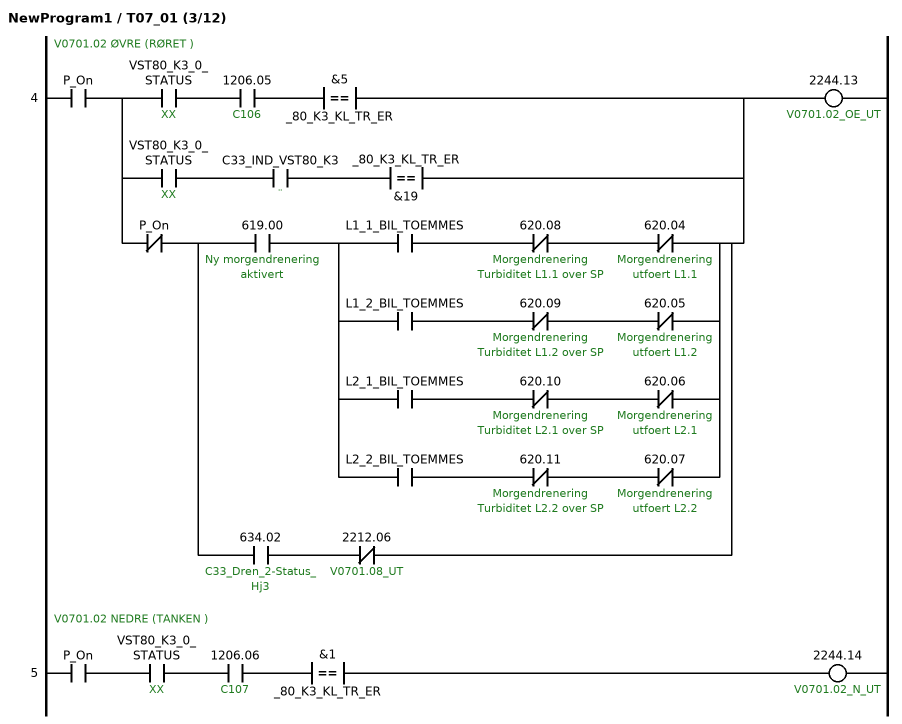
; rung 4: V0701.02 ØVRE (RØRET )
LD P_On
LD VST80_K3_0_STATUS  ; XX
AND 1206.05  ; C106
AND=(300) &5 _80_K3_KL_TR_ER
LD VST80_K3_0_STATUS  ; XX
AND C33_IND_VST80_K3  ; ¨
AND=(300) _80_K3_KL_TR_ER &19
ORLD
LDNOT P_On
LD 619.00  ; Ny morgendrenering aktivert
LD L1_1_BIL_TOEMMES
ANDNOT 620.08  ; Morgendrenering Turbiditet L1.1 over SP
ANDNOT 620.04  ; Morgendrenering utfoert L1.1
LD L1_2_BIL_TOEMMES
ANDNOT 620.09  ; Morgendrenering Turbiditet L1.2 over SP
ANDNOT 620.05  ; Morgendrenering utfoert L1.2
ORLD
LD L2_1_BIL_TOEMMES
ANDNOT 620.10  ; Morgendrenering Turbiditet L2.1 over SP
ANDNOT 620.06  ; Morgendrenering utfoert L2.1
ORLD
LD L2_2_BIL_TOEMMES
ANDNOT 620.11  ; Morgendrenering Turbiditet L2.2 over SP
ANDNOT 620.07  ; Morgendrenering utfoert L2.2
ORLD
ANDLD
LD 634.02  ; C33_Dren_2-Status_Hj3
ANDNOT 2212.06  ; V0701.08_UT
ORLD
ANDLD
ORLD
ANDLD
OUT 2244.13  ; V0701.02_OE_UT
; rung 5: V0701.02 NEDRE (TANKEN )
LD P_On
AND VST80_K3_0_STATUS  ; XX
AND 1206.06  ; C107
AND=(300) &1 _80_K3_KL_TR_ER
OUT 2244.14  ; V0701.02_N_UT

